Staubli VAL3: onStart.pgx

program onStart()
  local num i
begin
  // wait the START

end
